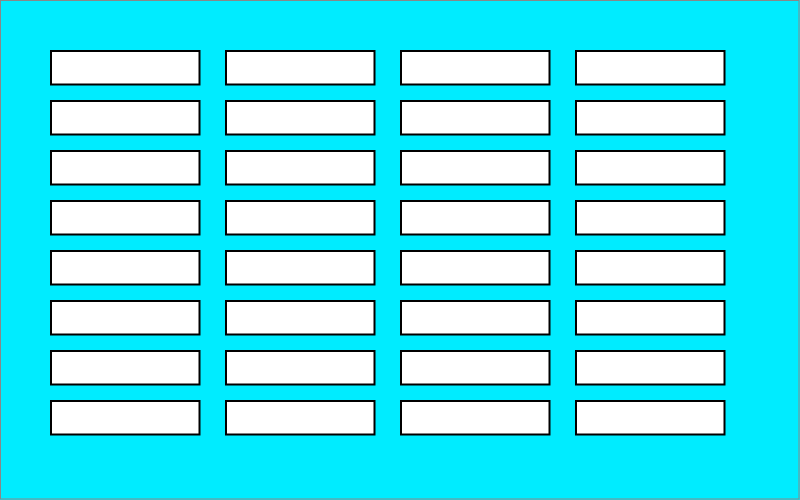
VISUALIZATION Screen_1_Sub_4  // 800x500
    Rectangle (0,0 800x500)
    Rectangle (50,50 150x35), "Val 1: %i", text variable: GVL.HMI_Number_Display[0]
    Rectangle (225,50 150x35), "Val 2: %i", text variable: GVL.HMI_Number_Display[1]
    Rectangle (400,50 150x35), "Val 3: %i", text variable: GVL.HMI_Number_Display[2]
    Rectangle (575,50 150x35), "Val 4: %i", text variable: GVL.HMI_Number_Display[3]
    Rectangle (50,100 150x35), "Val 5: %i", text variable: GVL.HMI_Number_Display[4]
    Rectangle (225,100 150x35), "Val 6: %i", text variable: GVL.HMI_Number_Display[5]
    Rectangle (400,100 150x35), "Val 7: %i", text variable: GVL.HMI_Number_Display[6]
    Rectangle (575,100 150x35), "Val 8: %i", text variable: GVL.HMI_Number_Display[7]
    Rectangle (50,150 150x35), "Val 9: %i", text variable: GVL.HMI_Number_Display[8]
    Rectangle (225,150 150x35), "Val 10: %i", text variable: GVL.HMI_Number_Display[9]
    Rectangle (400,150 150x35), "Val 11: %i", text variable: GVL.HMI_Number_Display[10]
    Rectangle (575,150 150x35), "Val 12: %i", text variable: GVL.HMI_Number_Display[11]
    Rectangle (50,200 150x35), "Val 13: %i", text variable: GVL.HMI_Number_Display[12]
    Rectangle (225,200 150x35), "Val 14: %i", text variable: GVL.HMI_Number_Display[13]
    Rectangle (400,200 150x35), "Val 15: %i", text variable: GVL.HMI_Number_Display[14]
    Rectangle (575,200 150x35), "Val 16: %i", text variable: GVL.HMI_Number_Display[15]
    Rectangle (50,250 150x35), "Val 17: %i", text variable: GVL.HMI_Number_Display[16]
    Rectangle (225,250 150x35), "Val 18: %i", text variable: GVL.HMI_Number_Display[17]
    Rectangle (400,250 150x35), "Val 19: %i", text variable: GVL.HMI_Number_Display[18]
    Rectangle (575,250 150x35), "Val 20: %i", text variable: GVL.HMI_Number_Display[19]
    Rectangle (50,300 150x35), "Val 21: %i", text variable: GVL.HMI_Number_Display[20]
    Rectangle (225,300 150x35), "Val 22: %i", text variable: GVL.HMI_Number_Display[21]
    Rectangle (400,300 150x35), "Val 23: %i", text variable: GVL.HMI_Number_Display[22]
    Rectangle (575,300 150x35), "Val 24: %i", text variable: GVL.HMI_Number_Display[23]
    Rectangle (50,350 150x35), "Val 25: %i", text variable: GVL.HMI_Number_Display[24]
    Rectangle (225,350 150x35), "Val 26: %i", text variable: GVL.HMI_Number_Display[25]
    Rectangle (400,350 150x35), "Val 27: %i", text variable: GVL.HMI_Number_Display[26]
    Rectangle (575,350 150x35), "Val 28: %i", text variable: GVL.HMI_Number_Display[27]
    Rectangle (50,400 150x35), "Val 29: %i", text variable: GVL.HMI_Number_Display[28]
    Rectangle (225,400 150x35), "Val 30: %i", text variable: GVL.HMI_Number_Display[29]
    Rectangle (400,400 150x35), "Val 31: %i", text variable: GVL.HMI_Number_Display[30]
    Rectangle (575,400 150x35), "Val 32: %i", text variable: GVL.HMI_Number_Display[31]
END_VISUALIZATION

(* stored: Version 1.1.0.1, ProductVersion 3.1.4024.12
   Visu Screen_1_Sub_4: Id {7cf601a0-c996-4b16-b60d-319a8db355dd} *)
